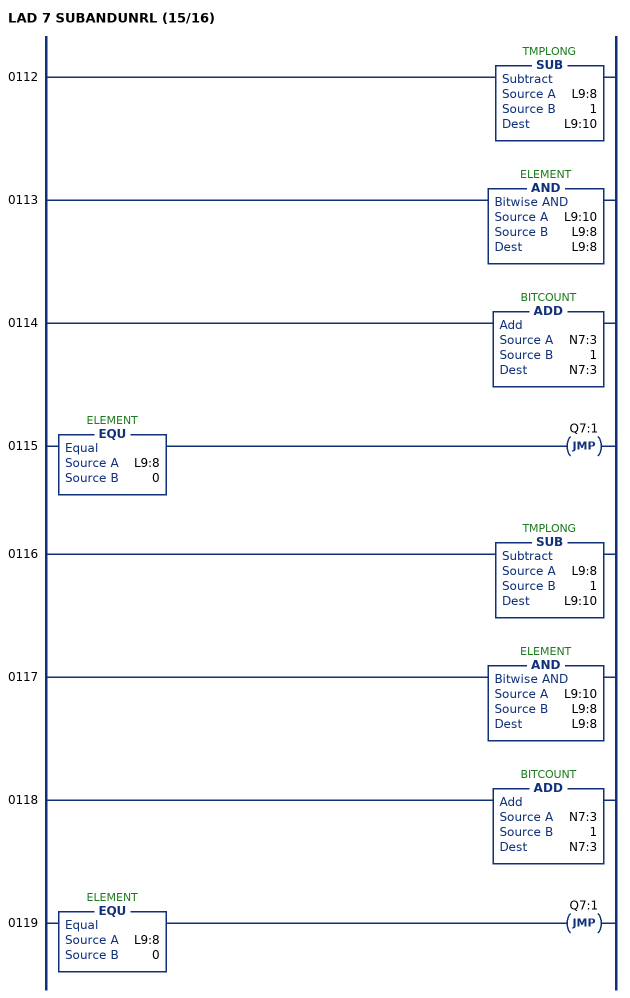
% Rung: 112 %
SOR SUB L9:8 1 L9:10 EOR
%   L9:8  ELEMENT %
%   L9:10  TMPLONG %
% Rung: 113 %
SOR AND L9:10 L9:8 L9:8 EOR
%   L9:10  TMPLONG %
%   L9:8  ELEMENT %
% Rung: 114 %
SOR ADD N7:3 1 N7:3 EOR
%   N7:3  BITCOUNT %
% Rung: 115 %
SOR EQU L9:8 0 JMP Q7:1 EOR
%   L9:8  ELEMENT %
% Rung: 116 %
SOR SUB L9:8 1 L9:10 EOR
%   L9:8  ELEMENT %
%   L9:10  TMPLONG %
% Rung: 117 %
SOR AND L9:10 L9:8 L9:8 EOR
%   L9:10  TMPLONG %
%   L9:8  ELEMENT %
% Rung: 118 %
SOR ADD N7:3 1 N7:3 EOR
%   N7:3  BITCOUNT %
% Rung: 119 %
SOR EQU L9:8 0 JMP Q7:1 EOR
%   L9:8  ELEMENT %

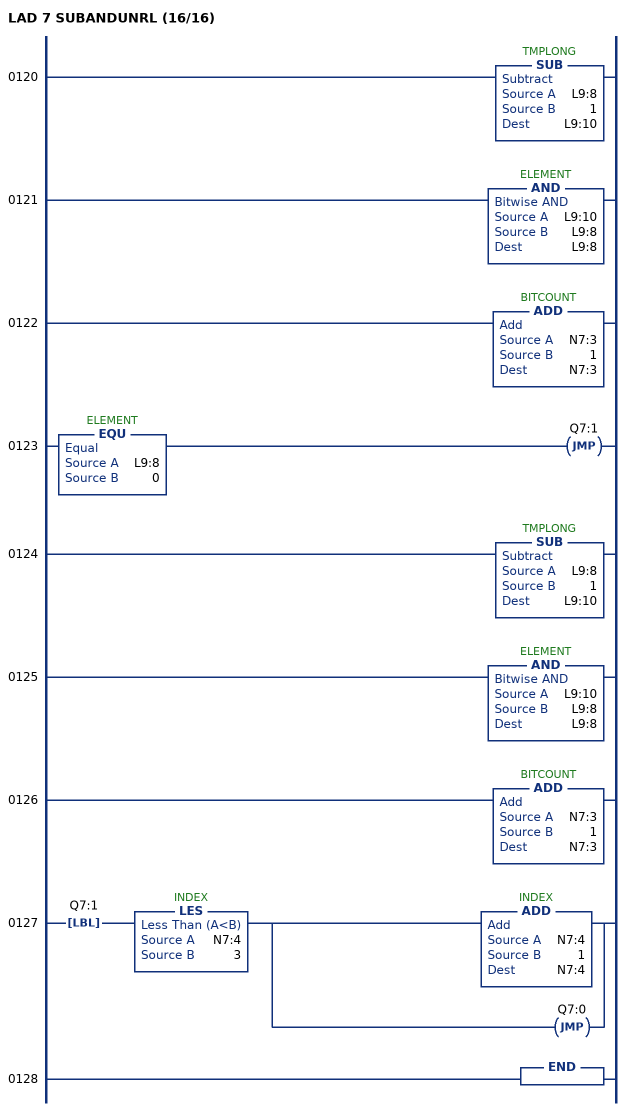
% Rung: 120 %
SOR SUB L9:8 1 L9:10 EOR
%   L9:8  ELEMENT %
%   L9:10  TMPLONG %
% Rung: 121 %
SOR AND L9:10 L9:8 L9:8 EOR
%   L9:10  TMPLONG %
%   L9:8  ELEMENT %
% Rung: 122 %
SOR ADD N7:3 1 N7:3 EOR
%   N7:3  BITCOUNT %
% Rung: 123 %
SOR EQU L9:8 0 JMP Q7:1 EOR
%   L9:8  ELEMENT %
% Rung: 124 %
SOR SUB L9:8 1 L9:10 EOR
%   L9:8  ELEMENT %
%   L9:10  TMPLONG %
% Rung: 125 %
SOR AND L9:10 L9:8 L9:8 EOR
%   L9:10  TMPLONG %
%   L9:8  ELEMENT %
% Rung: 126 %
SOR ADD N7:3 1 N7:3 EOR
%   N7:3  BITCOUNT %
% Rung: 127 %
SOR LBL Q7:1 LES N7:4 3 BST ADD N7:4 1 N7:4 NXB JMP Q7:0 BND EOR
%   N7:4  INDEX %
% Rung: 128 %
SOR END EOR

LADDER 254 "WRITE_BITS"
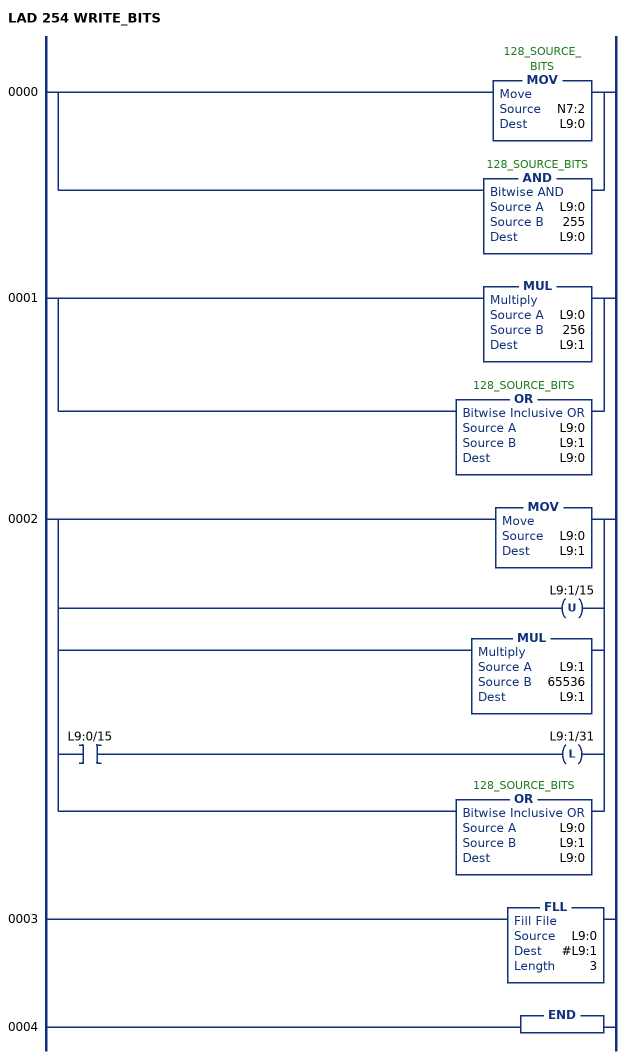
% Rung: 0 %
SOR BST MOV N7:2 L9:0 NXB AND L9:0 255 L9:0 BND EOR
%   N7:2  WHICH  "000-255:CONTROL ...-511:SUB/AND ...-767:PARALLEL ...-1023:XIC ...-1279:LOOKUP_BYTE" %
%   L9:0  128_SOURCE_BITS %
% Rung: 1 %
SOR BST MUL L9:0 256 L9:1 NXB OR L9:0 L9:1 L9:0 BND EOR
%   L9:0  128_SOURCE_BITS %
% Rung: 2 %
SOR BST MOV L9:0 L9:1 NXB OTU L9:1/15 NXB MUL L9:1 65536 L9:1 NXB XIC L9:0/15 OTL L9:1/31 NXB OR L9:0 L9:1 L9:0 BND EOR
%   L9:0  128_SOURCE_BITS %
% Rung: 3 %
SOR FLL L9:0 #L9:1 3 EOR
%   L9:0  128_SOURCE_BITS %
% Rung: 4 %
SOR END EOR

LADDER 255 "BITSPRBYTE"
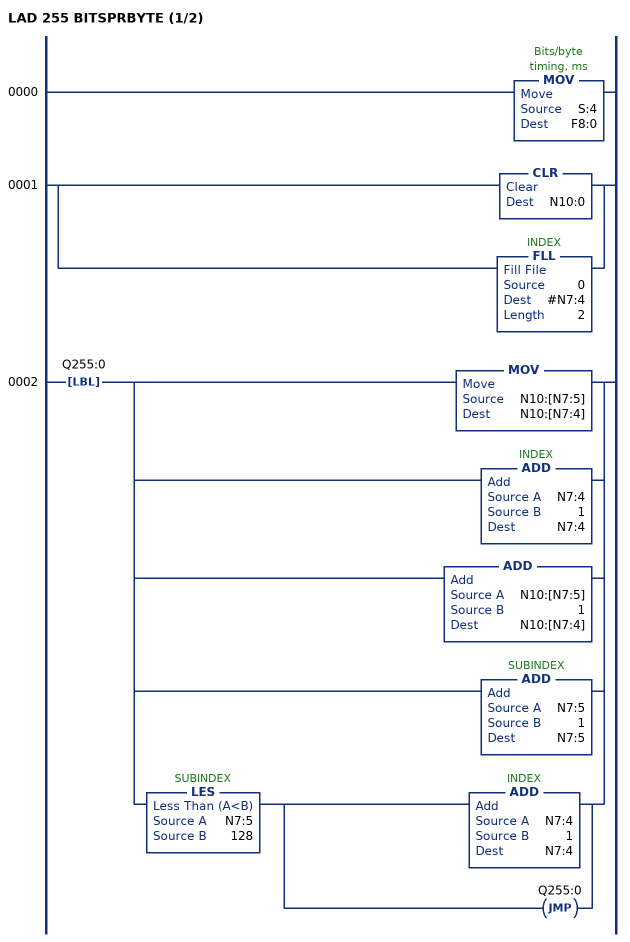
% Rung: 0 %
SOR MOV S:4 F8:0 EOR
%   S:4  "Time Base" %
%   F8:0  "Bits/byte timing, ms" %
% Rung: 1 %
SOR BST CLR N10:0 NXB FLL 0 #N7:4 2 BND EOR
%   N7:4  INDEX %
% Rung: 2 %
SOR LBL Q255:0 BST MOV N10:[N7:5] N10:[N7:4] NXB ADD N7:4 1 N7:4 NXB ADD N10:[N7:5] 1 N10:[N7:4] NXB ADD N7:5 1 N7:5 NXB LES N7:5 128 BST ADD N7:4 1 N7:4 NXB JMP Q255:0 BND BND EOR
%   N7:5  SUBINDEX %
%   N7:4  INDEX %

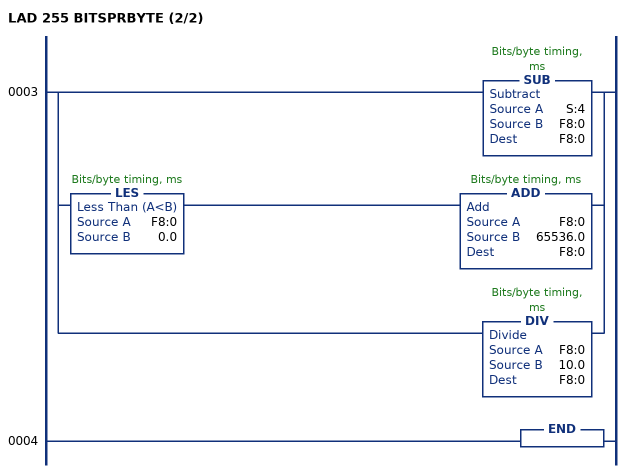
% Rung: 3 %
SOR BST SUB S:4 F8:0 F8:0 NXB LES F8:0 0.0 ADD F8:0 65536.0 F8:0 NXB DIV F8:0 10.0 F8:0 BND EOR
%   S:4  "Time Base" %
%   F8:0  "Bits/byte timing, ms" %
% Rung: 4 %
SOR END EOR

OTHER DOCUMENTED ADDRESSES
  L9:4  128_WORKING_BITS
  N7:6  8BITS

OTHER INSTRUCTION COMMENTS
  L9:4 NEQ  "First Working Long"

COMMENTS NOT ATTACHED TO A CURRENT RUNG
  N7:2/4: Restore preserved (cf. Rung 0005 above) bit values for /4 and /5

DATA TABLE (non-zero values as saved)
DATA T4
% .PRE .ACC %
% T4:1 % 5000 0
% T4:10 % 25 0
DATA C5
% .PRE .ACC %
% C5:0 % 1 0
DATA R6
% .LEN .POS %
% R6:0 % 128 0
DATA N7
% N7:0 % 1000 -1 0 0 0 0 0 0 0 0
DATA L9
% L9:5 % 0 0 0 0 32588
DATA L11
% L11:0 % 1431655765 858993459 252645135 16711935 65535
% L11:5 % -2 -4 -16 -256 -65536
